Fanuc KAREL source: PURGE_DEV.kl

PROGRAM T
%NOLOCKGROUP
VAR
 v0 : STRING[40]
 v1 : INTEGER
BEGIN
 PURGE_DEV(v0, v1)
END T
